# EPICS alarm handler configuration: alh_files/mgnt_in20Gs.alhConfig
GROUP NULL MGNT:IN20GS:1
   $COMMAND edm -x -eolc -noedit mgnt_in20_main.edl

$ALIAS IN20GS
$GUIDANCE
in20 Dog Leg Region
   Group Name: MGNT:IN20GS:1
   Summary PV:  MGNT:IN20GS:1:STATSUMY
$END

   INCLUDE MGNT:IN20GS:1 ./mgnt_in20Gs_bend.alhConfig
   INCLUDE MGNT:IN20GS:1 ./mgnt_in20Gs_lgps.alhConfig
   INCLUDE MGNT:IN20GS:1 ./mgnt_in20Gs_quad.alhConfig
   INCLUDE MGNT:IN20GS:1 ./mgnt_in20Gs_xcor.alhConfig
   INCLUDE MGNT:IN20GS:1 ./mgnt_in20Gs_ycor.alhConfig
